// TIA Portal V19 export
VAR_GLOBAL   // PLC tag table "04_SAFETY_SINAMICS_A03"
   NavettaAxTesta_StsIn AT %I1518.0 : "udt_LDrvSafe_typeSinaSTlg30Status";
   NavettaAxTesta_CtrlOut AT %Q1518.0 : "udt_LDrvSafe_typeSinaSTlg30Control";
   NavettaAxCoda_StsIn AT %I1528.0 : "udt_LDrvSafe_typeSinaSTlg30Status";
   NavettaAxCoda_CtrlOut AT %Q1528.0 : "udt_LDrvSafe_typeSinaSTlg30Control";
   RullieraAx1_StsIn AT %I968.0 : "udt_LDrvSafe_typeSinaSTlg30Status";
   RullieraAx1_CtrlOut AT %Q968.0 : "udt_LDrvSafe_typeSinaSTlg30Control";
   RullieraAx2_StsIn AT %I978.0 : "udt_LDrvSafe_typeSinaSTlg30Status";
   RullieraAx2_CtrlOut AT %Q978.0 : "udt_LDrvSafe_typeSinaSTlg30Control";
   PareggiatoreTestaAx_StsIn AT %I984.0 : "udt_LDrvSafe_typeSinaSTlg30Status";
   PareggiatoreTestaAx_CtrlOut AT %Q984.0 : "udt_LDrvSafe_typeSinaSTlg30Control";
   PareggiatoreCodaAx_StsIn AT %I990.0 : "udt_LDrvSafe_typeSinaSTlg30Status";
   PareggiatoreCodaAx_CtrlOut AT %Q990.0 : "udt_LDrvSafe_typeSinaSTlg30Control";
   ManipolatoreTestaAx_StsIn AT %I1380.0 : "udt_LDrvSafe_typeSinaSTlg30Status";
   ManipolatoreTestaAx_CtrlOut AT %Q1380.0 : "udt_LDrvSafe_typeSinaSTlg30Control";
   ManipolatoreCodaAx_StsIn AT %I1386.0 : "udt_LDrvSafe_typeSinaSTlg30Status";
   ManipolatoreCodaAx_CtrlOut AT %Q1386.0 : "udt_LDrvSafe_typeSinaSTlg30Control";
   SpallaCodaAx_StsIn AT %I1350.0 : "udt_LDrvSafe_typeSinaSTlg30Status";
   SpallaCodaAx_CtrlOut AT %Q1350.0 : "udt_LDrvSafe_typeSinaSTlg30Control";
   SpallaTestaAx_StsIn AT %I1344.0 : "udt_LDrvSafe_typeSinaSTlg30Status";
   SpallaTestaAx_CtrlOut AT %Q1344.0 : "udt_LDrvSafe_typeSinaSTlg30Control";
   TraslazioneTestaAx_StsIn AT %I1280.0 : "udt_LDrvSafe_typeSinaSTlg30Status";
   TraslazioneTestaAx_CtrlOut AT %Q1280.0 : "udt_LDrvSafe_typeSinaSTlg30Control";
   TraslazioneCodaAx_StsIn AT %I1286.0 : "udt_LDrvSafe_typeSinaSTlg30Status";
   TraslazioneCodaAx_CtrlOut AT %Q1286.0 : "udt_LDrvSafe_typeSinaSTlg30Control";
   SostegnoAntiribCodaAx_StsIn AT %I1548.0 : "udt_LDrvSafe_typeSinaSTlg30Status";
   SostegnoAntiribCodaAx_CtrlOut AT %Q1548.0 : "udt_LDrvSafe_typeSinaSTlg30Control";
   SostegnoAntiribTestaAx_StsIn AT %I1538.0 : "udt_LDrvSafe_typeSinaSTlg30Status";
   SostegnoAntiribTestaAx_CtrlOut AT %Q1538.0 : "udt_LDrvSafe_typeSinaSTlg30Control";
   SollevamentoTestaAx_StsIn AT %I1392.0 : "udt_LDrvSafe_typeSinaSTlg30Status";
   SollevamentoTestaAx_CtrlOut AT %Q1392.0 : "udt_LDrvSafe_typeSinaSTlg30Control";
   SollevamentoCodaAx_StsIn AT %I1512.0 : "udt_LDrvSafe_typeSinaSTlg30Status";
   SollevamentoCodaAx_CtrlOut AT %Q1512.0 : "udt_LDrvSafe_typeSinaSTlg30Control";
   BordatriceAx_StsIn AT %I832.0 : "udt_LDrvSafe_typeSinaSTlg30Status";
   BordatriceAx_CtrlOut AT %Q832.0 : "udt_LDrvSafe_typeSinaSTlg30Control";
   RibaltatoreAx_StsIn AT %I882.0 : "udt_LDrvSafe_typeSinaSTlg30Status";
   RibaltatoreAx_CtrlOut AT %Q882.0 : "udt_LDrvSafe_typeSinaSTlg30Control";
   SpintoreAx_StsIn AT %I888.0 : "udt_LDrvSafe_typeSinaSTlg30Status";
   SpintoreAx_CtrlOut AT %Q888.0 : "udt_LDrvSafe_typeSinaSTlg30Control";
   TrasportoAx_StsIn AT %I842.0 : "udt_LDrvSafe_typeSinaSTlg30Status";
   TrasportoAx_CtrlOut AT %Q842.0 : "udt_LDrvSafe_typeSinaSTlg30Control";
   BordatriceCassettaAx_StsIn AT %I1065.0 : "udt_LDrvSafe_typeSinaSTlg30Control";
   BordatriceCassettaAx_CtrlOut AT %Q1065.0 : "udt_LDrvSafe_typeSinaSTlg30Control";
END_VAR
